(* PLC project Unnamed, Unknown Unnamed 1 *)
(* stored: creationDateTime 2022-12-13T19:44:02, modificationDateTime 2023-01-02T17:10:47 *)

PROGRAM water_tank
  VAR
    Valve_In AT %QX0.0 : BOOL;
    Valve_Out AT %QX0.1 : BOOL;
    Start AT %QX0.2 : BOOL;
    Stop AT %QX0.3 : BOOL;
    High AT %IX0.0 : BOOL;
    Low AT %IX0.1 : BOOL;
    Master AT %IX0.2 : BOOL;
    Height_In AT %IW0 : UINT;
    Height_Out AT %QW0 : UINT;
    High_Limit AT %QW1 : UINT;
    Low_Limit AT %QW2 : UINT;
  END_VAR

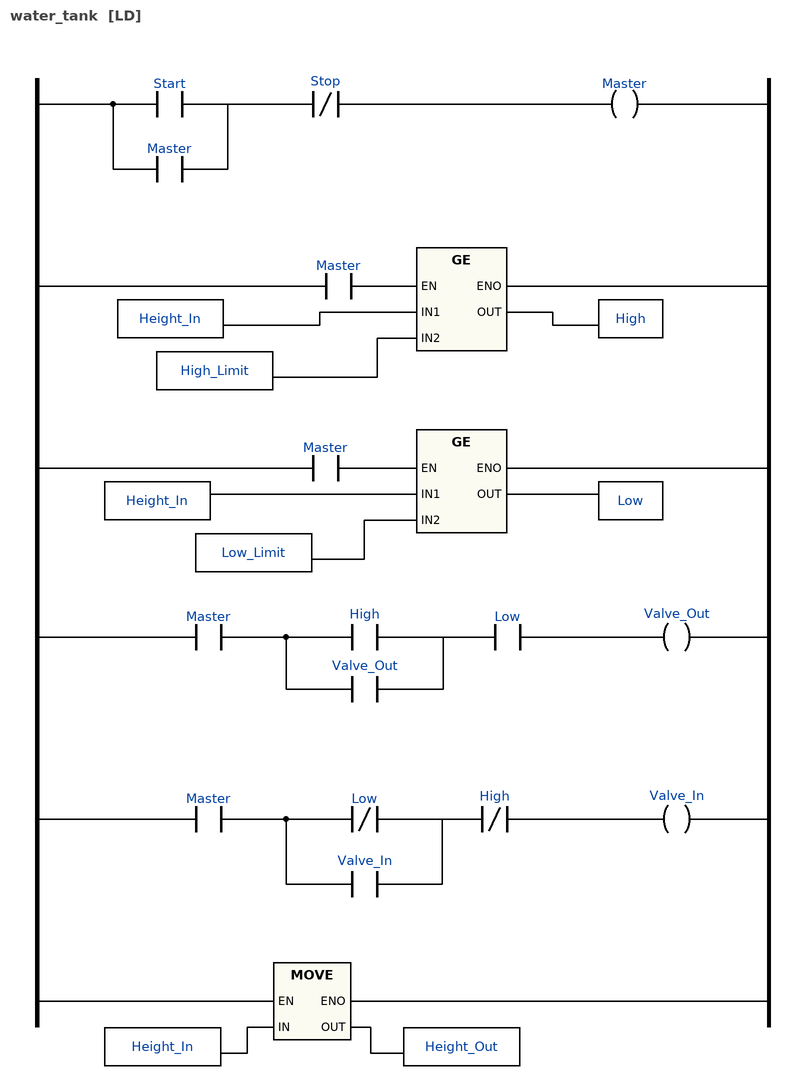
(* LD diagram, written out as Structured Text *)
Master := (Start OR Master) AND NOT Stop;
IF Master THEN High := Height_In >= High_Limit; END_IF;
IF Master THEN Low := Height_In >= Low_Limit; END_IF;
Valve_Out := Master AND (High OR Valve_Out) AND Low;
Valve_In := Master AND (NOT Low OR Valve_In) AND NOT High;
Height_Out := Height_In;
END_PROGRAM

CONFIGURATION Config0
  RESOURCE Res0 ON PLC
    TASK task0(INTERVAL := T#20ms, PRIORITY := 0);
    PROGRAM instance0 WITH task0 : water_tank;
  END_RESOURCE
END_CONFIGURATION
